(* Visualisation AUTO1
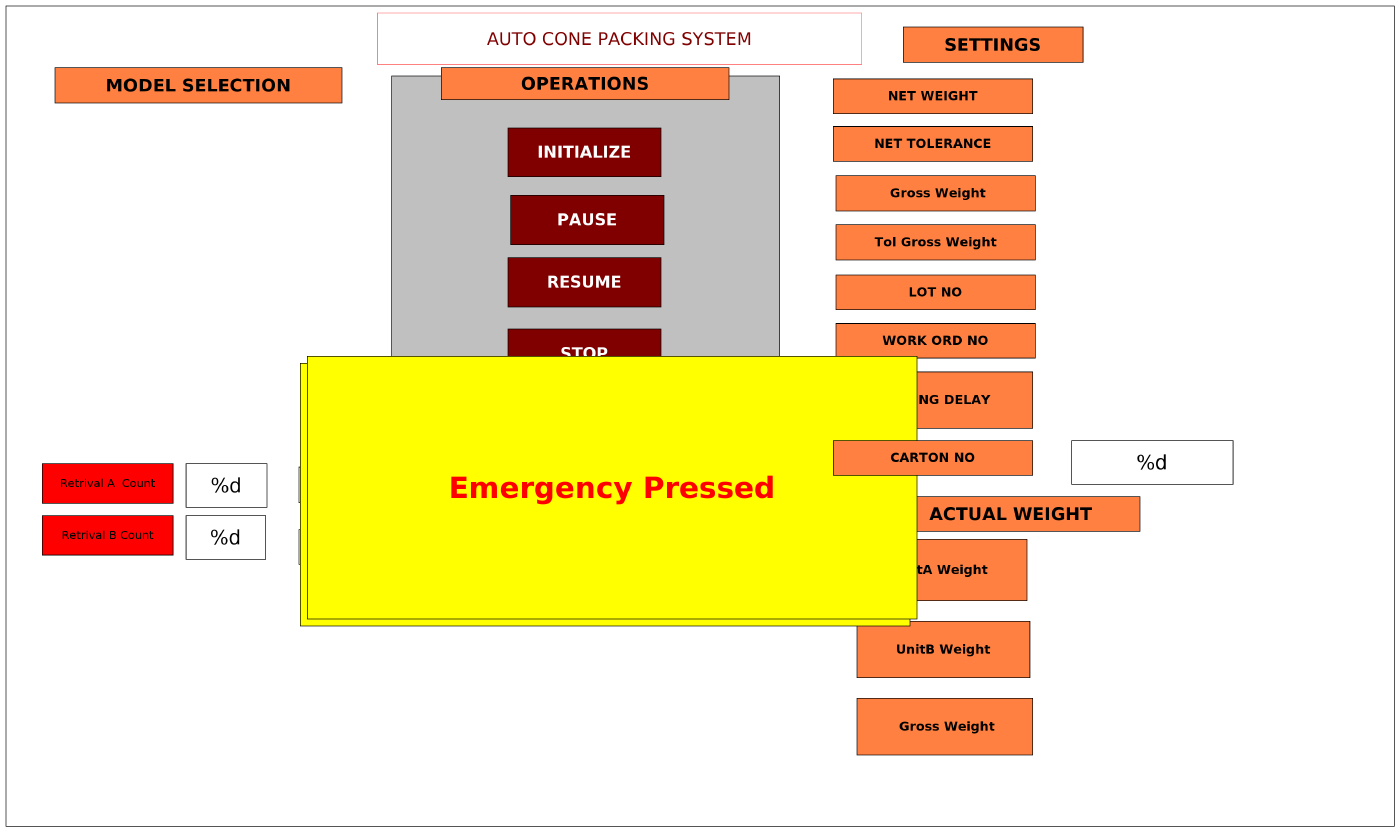
rounded rectangle at (530,10)-(1221,84): text "AUTO CONE PACKING SYSTEM"
rounded rectangle at (418,658)-(674,709): text "Machine Status"
rounded rectangle at (693,648)-(1093,718): text "%s"; shows sAMcModeStatus
rounded rectangle at (418,747)-(674,797): text "Alarm Status"
rounded rectangle at (693,737)-(1093,807): text "%s"; shows sAlarmStatus
rounded rectangle at (70,88)-(480,139): text "MODEL SELECTION"
rounded rectangle at (1210,761)-(1457,849): text "UnitA Weight"
rounded rectangle at (1214,878)-(1461,959): text "UnitB Weight"
rounded rectangle at (1184,522)-(1465,603): text "SEALING DELAY"
rounded rectangle at (1280,30)-(1537,81): text "SETTINGS"
rounded rectangle at (1180,104)-(1465,154): text "NET WEIGHT"
rounded rectangle at (1180,172)-(1465,222): text "NET TOLERANCE"
rounded rectangle at (1249,700)-(1618,750): text "ACTUAL WEIGHT"
rounded rectangle at (257,727)-(371,790): text "%d"; shows UnitBConeCountHMI
rounded rectangle at (257,653)-(373,716): text "%d"; shows UnitAConeCountHMI
rectangle at (52,653)-(239,710): text "Retrival A  Count"
rectangle at (52,727)-(239,784): text "Retrival B Count"
rounded rectangle at (1184,384)-(1469,434): text "LOT NO"
rounded rectangle at (1184,242)-(1469,293): text "Gross Weight"
rounded rectangle at (1214,988)-(1465,1069): text "Gross Weight"
rounded rectangle at (1184,312)-(1469,363): text "Tol Gross Weight"
rounded rectangle at (1184,453)-(1469,503): text "WORK ORD NO"
rounded rectangle at (716,461)-(935,532): text "STOP"; alarm colour if bStopHmi; taps bStopHmi
rounded rectangle at (716,359)-(935,430): text "RESUME"; alarm colour if bAPauseSeq; taps bResumeHmi
rounded rectangle at (720,270)-(939,341): text "PAUSE"; alarm colour if bAPauseSeq; taps bPauseHmi
rounded rectangle at (716,174)-(935,244): text "INITIALIZE"; alarm colour if bAInitializeSeq; taps bInitializeHmi
rounded rectangle at (621,88)-(1032,134): text "OPERATIONS"
rounded rectangle at (420,510)-(1290,885): text "Supply Pressure Low"; invisible if NOT bPrssurePopUp
rounded rectangle at (430,500)-(1300,875): text "Emergency Pressed"; invisible if NOT bEmPopUp
rounded rectangle at (1180,620)-(1465,670): text "CARTON NO"
rounded rectangle at (1520,620)-(1751,683): text "%d"; shows CARTONNO_DIS
2 more shapes without text or variables
20 elements of other kinds (tables, trends, ...) not read
*)

(* Visualisation DIAGNOSTICS
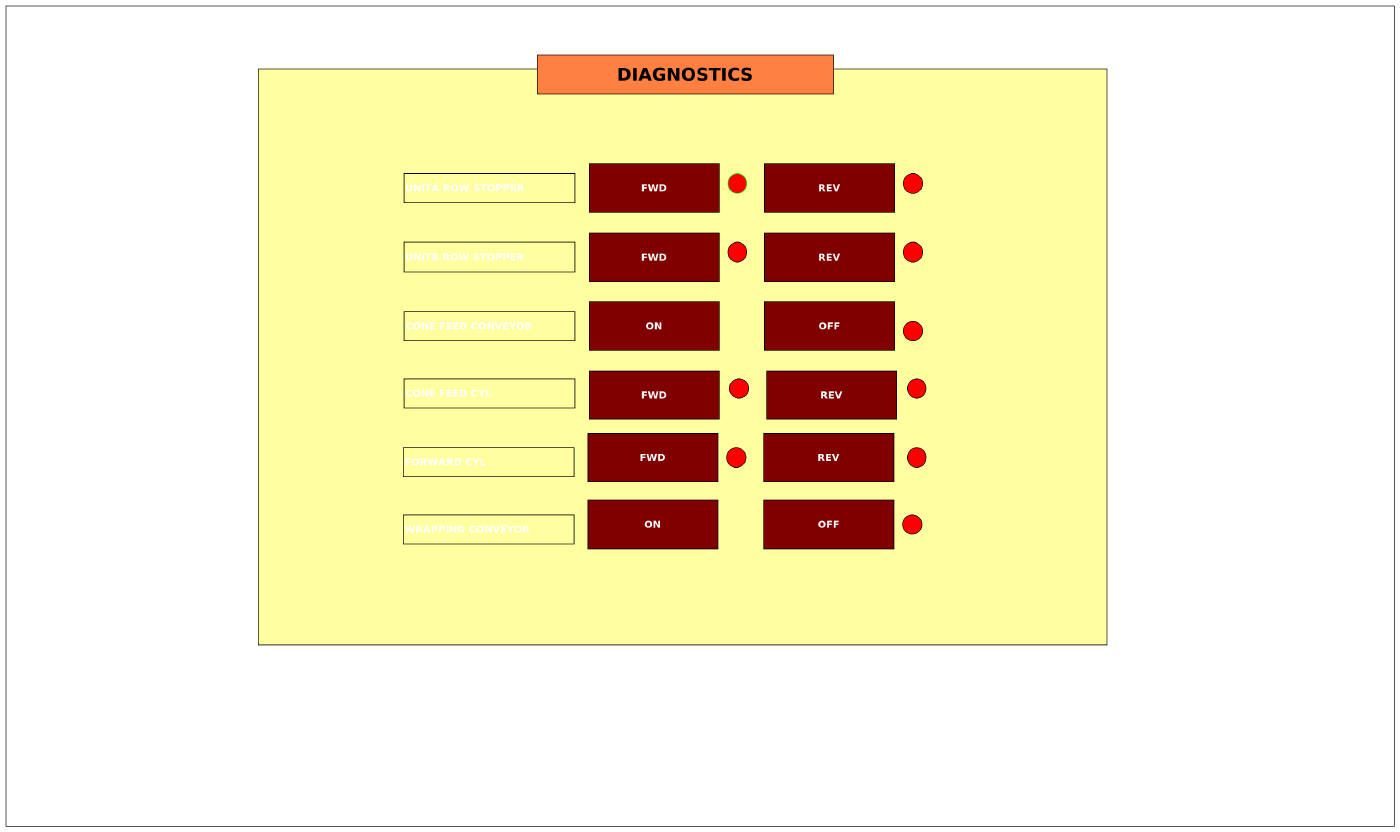
rounded rectangle at (758,70)-(1181,126): text "DIAGNOSTICS"
ellipse at (1030,239)-(1057,268): alarm colour if .bIUnitA_RowStopperEnd
ellipse at (1030,337)-(1057,366): alarm colour if .bIUnitB_RowStopperEnd
ellipse at (1280,239)-(1308,268): alarm colour if .bIUnitA_RowStopperHome
ellipse at (1280,337)-(1308,366): alarm colour if .bIUnitB_RowStopperHome
ellipse at (1280,450)-(1308,478): alarm colour if .bQFeedingConveyorMotor
rounded rectangle at (832,225)-(1018,295): text "FWD"; alarm colour if .bUA_RowStopperMotorFwdOnHmi; taps .bUA_RowStopperMotorFwdOnHmi
rounded rectangle at (1082,225)-(1268,295): text "REV"; alarm colour if .bUA_RowStopperMotorRevOnHmi; taps .bUA_RowStopperMotorRevOnHmi
rounded rectangle at (832,324)-(1018,394): text "FWD"; alarm colour if .bUB_RowStopperMotorFwdOnHmi; taps .bUB_RowStopperMotorFwdOnHmi
rounded rectangle at (832,422)-(1018,492): text "ON"; alarm colour if bFCMotorOnHmi; taps bFCMotorOnHmi
rounded rectangle at (1082,324)-(1268,394): text "REV"; alarm colour if .bUB_RowStopperMotorRevOnHmi; taps .bUB_RowStopperMotorRevOnHmi
rounded rectangle at (1082,422)-(1268,492): text "OFF"; alarm colour if bFCMotorOffHmi; taps bFCMotorOffHmi
rounded rectangle at (568,239)-(812,281): text "UNITA ROW STOPPER"
rounded rectangle at (568,337)-(812,380): text "UNITB ROW STOPPER"
rounded rectangle at (568,436)-(812,478): text "CONE FEED CONVEYOR"
ellipse at (1032,532)-(1060,560): alarm colour if .bIConeFeedingPistonEnd
ellipse at (1286,532)-(1313,560): alarm colour if .bIConeFeedingPistonHome
rounded rectangle at (832,521)-(1018,590): text "FWD"; alarm colour if .bCFPistonOnHmi; taps .bCFPistonOnHmi
rounded rectangle at (1085,521)-(1271,590): text "REV"; alarm colour if .bCFPistonOffHmi; taps .bCFPistonOffHmi
rounded rectangle at (568,532)-(812,574): text "CONE FEED CYL"
ellipse at (1279,726)-(1307,754): alarm colour if .bQMWrappingConveyorMotor
rounded rectangle at (830,705)-(1016,775): text "ON"; alarm colour if .bWCMotorOnHmi; taps .bWCMotorOnHmi
rounded rectangle at (1081,705)-(1267,775): text "OFF"; alarm colour if .bWCMotorOffHmi; taps .bWCMotorOffHmi
rounded rectangle at (567,726)-(811,768): text "WRAPPING CONVEYOR"
rounded rectangle at (567,630)-(811,672): text "FORWARD CYL"
rounded rectangle at (830,610)-(1016,679): text "FWD"; alarm colour if .bFPValveOnHmi; taps .bFPValveOnHmi
rounded rectangle at (1081,610)-(1267,679): text "REV"; alarm colour if .bFPValveOffHmi; taps .bFPValveOffHmi
ellipse at (1028,630)-(1056,659): alarm colour if .bIForwardPistonEnd
ellipse at (1286,630)-(1313,659): alarm colour if .bIForwardPistonHome
2 more shapes without text or variables
2 elements of other kinds (tables, trends, ...) not read
*)

(* Visualisation DIAGNOSTICS_1
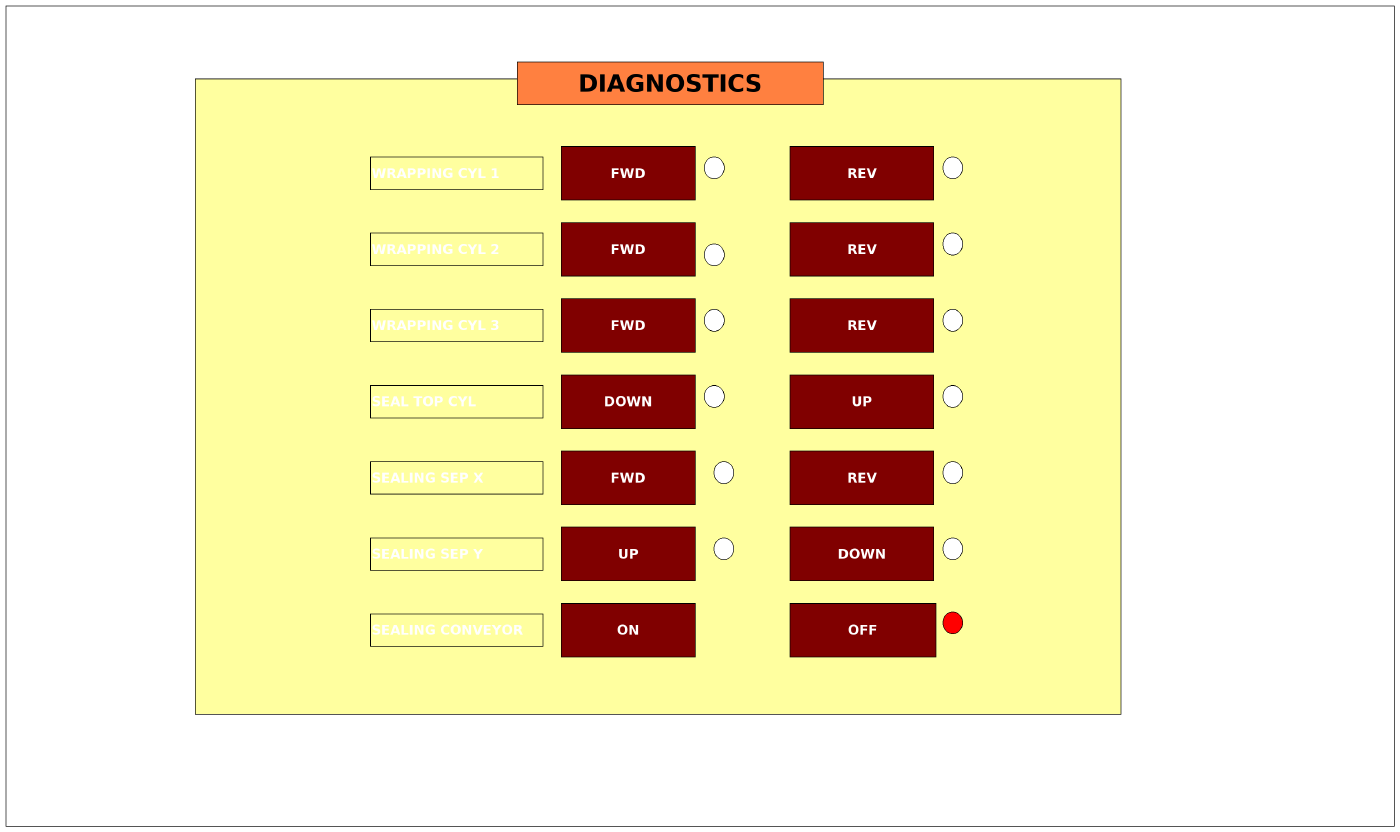
group at (270,80)-(1591,1011)
  rounded rectangle at (338,0)-(659,41): text "DIAGNOSTICS"
  rounded rectangle at (384,80)-(525,131): text "FWD"; alarm colour if .bWrappingCPV1OnHmi; taps .bWrappingCPV1OnHmi
  rounded rectangle at (384,152)-(525,203): text "FWD"; alarm colour if .bWrappingCPV2OnHmi; taps .bWrappingCPV2OnHmi
  rounded rectangle at (624,152)-(775,203): text "REV"; alarm colour if .bWrappingCPV2OffHmi; taps .bWrappingCPV2OffHmi
  rounded rectangle at (384,224)-(525,275): text "FWD"; alarm colour if .bWrappingCPV3OnHmi; taps .bWrappingCPV3OnHmi
  rounded rectangle at (624,224)-(775,275): text "REV"; alarm colour if .bWrappingCPV3OffHmi; taps .bWrappingCPV3OffHmi
  rounded rectangle at (384,296)-(525,347): text "DOWN"; alarm colour if .bSealingTopPVOnHmi; taps .bSealingTopPVOnHmi
  rounded rectangle at (624,296)-(775,347): text "UP"; alarm colour if bSealingTopPVOffHmi; taps bSealingTopPVOffHmi
  rounded rectangle at (384,368)-(525,419): text "FWD"; alarm colour if bSSXAxisPistonValveOnHmi; taps bSSXAxisPistonValveOnHmi
  rounded rectangle at (624,368)-(775,419): text "REV"; alarm colour if bSSXAxisPistonValveOffHmi; taps bSSXAxisPistonValveOffHmi
  rounded rectangle at (184,90)-(365,121): text "WRAPPING CYL 1"
  rounded rectangle at (184,162)-(365,193): text "WRAPPING CYL 2"
  rounded rectangle at (184,234)-(365,265): text "WRAPPING CYL 3"
  rounded rectangle at (184,306)-(365,337): text "SEAL TOP CYL"
  rounded rectangle at (184,378)-(365,409): text "SEALING SEP X"
  rounded rectangle at (624,80)-(775,131): text "REV"; alarm colour if .bWrappingCPV1OffHmi; taps .bWrappingCPV1OffHmi
  ellipse at (784,520)-(805,541): alarm colour if .bQMWrappingConveyorMotor
  rounded rectangle at (384,512)-(525,563): text "ON"; alarm colour if bSCMotorOnHmi; taps bSCMotorOnHmi
  rounded rectangle at (624,512)-(777,563): text "OFF"; alarm colour if bSCMotorOffHmi; taps bSCMotorOffHmi
  rounded rectangle at (184,522)-(365,553): text "SEALING CONVEYOR"
  rounded rectangle at (384,440)-(525,491): text "UP"; alarm colour if bSSYAxisPistonValveOnHmi; taps bSSYAxisPistonValveOnHmi
  rounded rectangle at (624,440)-(775,491): text "DOWN"; alarm colour if bSSYAxisPistonValveOffHmi; taps bSSYAxisPistonValveOffHmi
  rounded rectangle at (184,450)-(365,481): text "SEALING SEP Y"
14 more shapes without text or variables
*)

(* Visualisation OVERVIEW
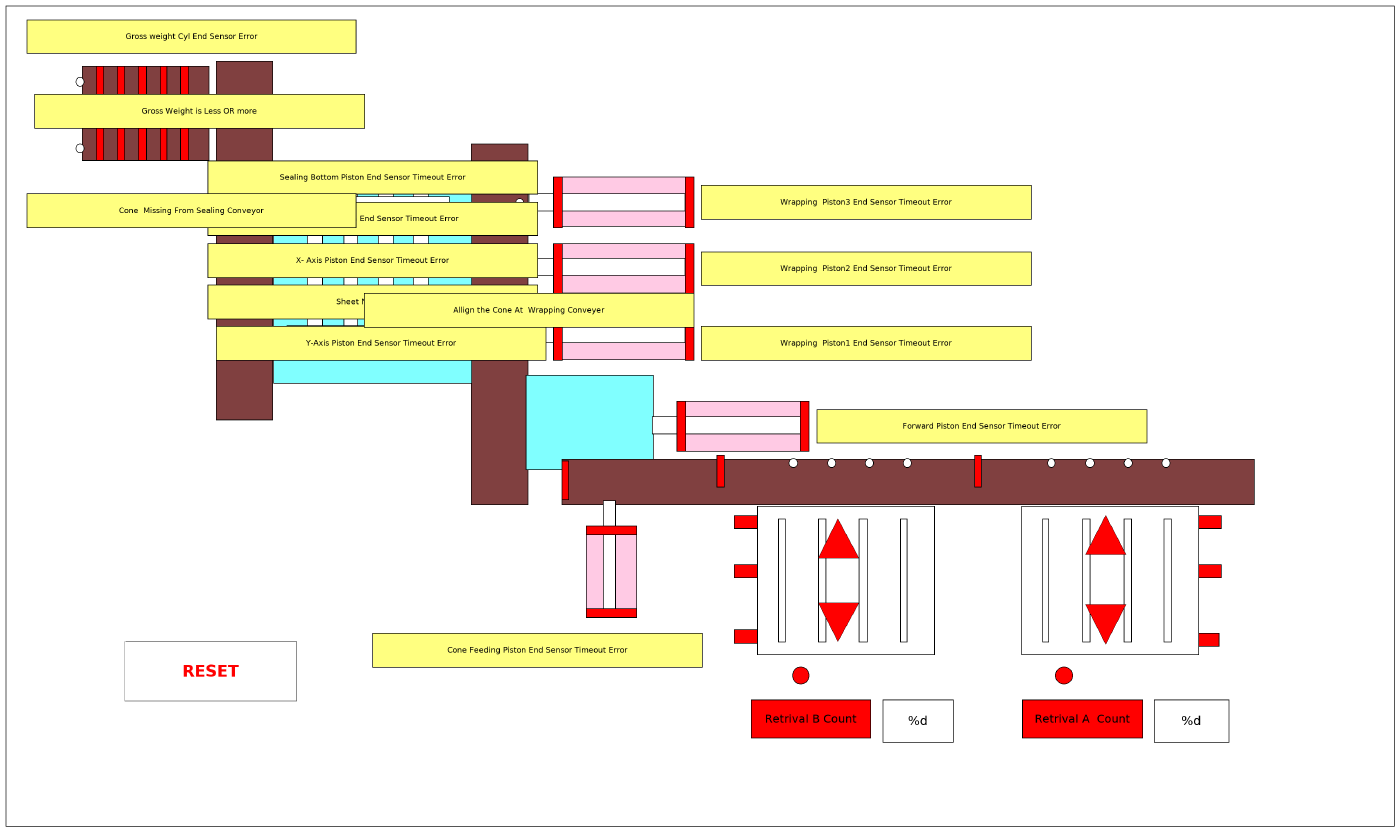
rectangle at (746,360)-(969,385): alarm colour if bQWrappingChannelPistonValve2
rectangle at (781,339)-(794,411): alarm colour if bIWrappingChannelPiston2_End
rectangle at (969,339)-(982,411): alarm colour if bIWrappingChannelPiston2_Home
rectangle at (1685,895)-(1731,914): alarm colour if bIUnitA_RowStopperHome
rectangle at (1692,797)-(1734,816): alarm colour if bIUnitA_RowStopperMiddle
rectangle at (1692,727)-(1734,746): alarm colour if bIUnitA_RowStopperEnd
rectangle at (1039,727)-(1077,746): alarm colour if bIUnitB_RowStopperEnd
rectangle at (1039,890)-(1077,910): alarm colour if bIUnitB_RowStopperHome
rectangle at (1039,797)-(1077,816): alarm colour if bIUnitB_RowStopperMiddle
rounded rectangle at (664,197)-(745,712): alarm colour if bQWrappingConveyorMotor
rectangle at (922,586)-(1144,611): alarm colour if bQForwardPistonValve
rounded rectangle at (793,647)-(1781,712): alarm colour if bQFeedingConveyorMotor
polygon at (1159,852)-(1217,907): alarm colour if bQUnitBRowStopperMotorRev
polygon at (1159,732)-(1217,788): alarm colour if bQUnitBRowStopperMotorFwd
polygon at (1540,854)-(1598,911): alarm colour if bQUnitARowStopperMotorRev
polygon at (1540,727)-(1598,783): alarm colour if bQUnitARowStopperMotorFwd
rectangle at (793,649)-(803,705): alarm colour if bIConeOrientationTop
rectangle at (1014,641)-(1025,687): alarm colour if bIUnitBConeCrossing
rectangle at (1382,641)-(1392,687): alarm colour if bIUnitAConeCrossing
rectangle at (852,706)-(870,872): alarm colour if bQConeFeedingPistonValve
rectangle at (746,457)-(969,481): alarm colour if bQWrappingChannelPistonValve1
rectangle at (746,268)-(969,293): alarm colour if bQWrappingChannelPistonValve3
rectangle at (482,240)-(502,488): alarm colour if bQSealingBottomPistonValve
rectangle at (430,240)-(452,488): alarm colour if bQSealingSeparatorXAxisPistonValve
rectangle at (531,240)-(553,488): alarm colour if bQSealingTopPistonValve
rectangle at (581,244)-(603,494): alarm colour if bQSealingSeparatorYAxisPistonValve
rounded rectangle at (300,79)-(381,591): alarm colour if bQSealingConveyorMotorFWD
rectangle at (109,86)-(290,221): alarm colour if bQGross_Cylinder_On
rectangle at (220,86)-(230,221): alarm colour if bQGross_Roller_On
rectangle at (249,86)-(261,221): alarm colour if bQGross_Roller_On
rectangle at (189,86)-(201,221): alarm colour if bQGross_Roller_On
rectangle at (159,86)-(170,221): alarm colour if bQGross_Roller_On
rectangle at (129,86)-(140,221): alarm colour if bQGross_Roller_On
rectangle at (401,456)-(633,478): alarm colour if bQFilmRollerMotor1
rectangle at (401,272)-(633,292): alarm colour if bQFilmRollerMotor3
rectangle at (401,363)-(633,385): alarm colour if bQFilmRollerMotor2
ellipse at (1540,646)-(1553,659): alarm colour if bIUnitAConeDetection3
ellipse at (1595,646)-(1607,659): alarm colour if bIUnitAConeDetection2
ellipse at (1649,646)-(1661,659): alarm colour if bIUnitAConeDetection1
ellipse at (1486,646)-(1497,659): alarm colour if bIUnitAConeDetection4
ellipse at (1172,646)-(1184,659): alarm colour if bIUnitBConeDetection3
ellipse at (1226,646)-(1238,659): alarm colour if bIUnitBConeDetection2
ellipse at (1280,646)-(1292,659): alarm colour if bIUnitBConeDetection1
ellipse at (1117,646)-(1130,659): alarm colour if bIUnitBConeDetection4
ellipse at (727,275)-(739,288): alarm colour if bIWrappingCone3
ellipse at (727,368)-(739,381): alarm colour if bIWrappingCone2
ellipse at (722,457)-(734,470): alarm colour if bIWrappingCone1
ellipse at (327,229)-(338,241): alarm colour if bIConeCountSensor
ellipse at (597,221)-(608,233): alarm colour if bISealingSeparatorYAxisEnd
ellipse at (441,221)-(453,233): alarm colour if bISealingSeparatorXAxisEnd
ellipse at (553,221)-(565,233): alarm colour if bISealingTopPistonEnd
ellipse at (499,221)-(511,233): alarm colour if bISealingBottomPistonEnd
ellipse at (100,102)-(112,115): alarm colour if bIGross_Cyl_Home
ellipse at (100,197)-(112,210): alarm colour if bIGross_Cyl_End
ellipse at (1122,943)-(1146,968): alarm colour if bQUnitBWeightOkLamp
ellipse at (1497,943)-(1522,968): alarm colour if bQUnitAWeightOkLamp
rectangle at (781,244)-(794,317): alarm colour if bIWrappingChannelPiston3_End
rectangle at (969,244)-(982,317): alarm colour if bIWrappingChannelPiston3_Home
rectangle at (781,434)-(794,506): alarm colour if bIWrappingChannelPiston1_End
rectangle at (969,434)-(982,506): alarm colour if bIWrappingChannelPiston1_Home
rectangle at (828,742)-(900,755): alarm colour if bIConeFeedingPistonEnd
rectangle at (828,860)-(900,873): alarm colour if bIConeFeedingPistonHome
rectangle at (1133,564)-(1146,636): alarm colour if bIForwardPistonHome
ellipse at (592,493)-(605,506): alarm colour if bISealingSeparatorYAxisHome
ellipse at (441,493)-(452,506): alarm colour if bISealingSeparatorXAxisHome
ellipse at (549,493)-(561,506): alarm colour if bISealingTopPistonHome
ellipse at (495,493)-(506,506): alarm colour if bISealingBottomPistonHome
rectangle at (523,895)-(994,944): text "Cone Feeding Piston End Sensor Timeout Error"; invisible if NOT bAConeFeedCylRsError
rectangle at (992,457)-(1463,506): text "Wrapping  Piston1 End Sensor Timeout Error"; invisible if NOT bAWrappingCylRs1Error
rectangle at (992,256)-(1463,305): text "Wrapping  Piston3 End Sensor Timeout Error"; invisible if NOT bAWrappingCylRs3Error
rectangle at (992,351)-(1463,399): text "Wrapping  Piston2 End Sensor Timeout Error"; invisible if NOT bAWrappingCylRs2Error
rectangle at (288,221)-(759,269): text "Sealing Bottom Piston End Sensor Timeout Error"; invisible if NOT bASealBotCylRsError
rectangle at (288,280)-(759,328): text "Sealing Top Piston End Sensor Timeout Error"; invisible if NOT bASealTopCylRsError
rectangle at (288,339)-(759,388): text "X- Axis Piston End Sensor Timeout Error"; invisible if NOT bASealSepXCylRsError
rectangle at (300,457)-(771,506): text "Y-Axis Piston End Sensor Timeout Error"; invisible if NOT bASealSepYCylRsError
rectangle at (288,398)-(759,447): text "Sheet NOT Feeded"; invisible if NOT bAPolythinSheetError
rectangle at (30,268)-(500,317): text "Cone  Missing From Sealing Conveyor"; invisible if NOT bAConeMissAtSealConv
rectangle at (511,410)-(982,459): text "Allign the Cone At  Wrapping Conveyer"; invisible if NOT bAConeMissErrorAtWrpConv
rectangle at (41,126)-(512,175): text "Gross Weight is Less OR more"; invisible if NOT bGrossWieghtNOk
rectangle at (1157,576)-(1628,624): text "Forward Piston End Sensor Timeout Error"; invisible if NOT bAFwdCylRsError
rectangle at (30,20)-(500,68): text "Gross weight Cyl End Sensor Error"; invisible if NOT bGrossWtCylEndSenError
button at (170,907)-(415,992): text "RESET"; shows .bErrorReset; taps .bErrorResethmi
rounded rectangle at (1251,990)-(1352,1051): text "%d"; shows UnitBConeCountHMI
rounded rectangle at (1638,990)-(1745,1051): text "%d"; shows UnitAConeCountHMI_1
rectangle at (1450,990)-(1622,1045): text "Retrival A  Count"
rectangle at (1063,990)-(1234,1045): text "Retrival B Count"
19 more shapes without text or variables
6 elements of other kinds (tables, trends, ...) not read
*)

(* Visualisation PARAMETERS
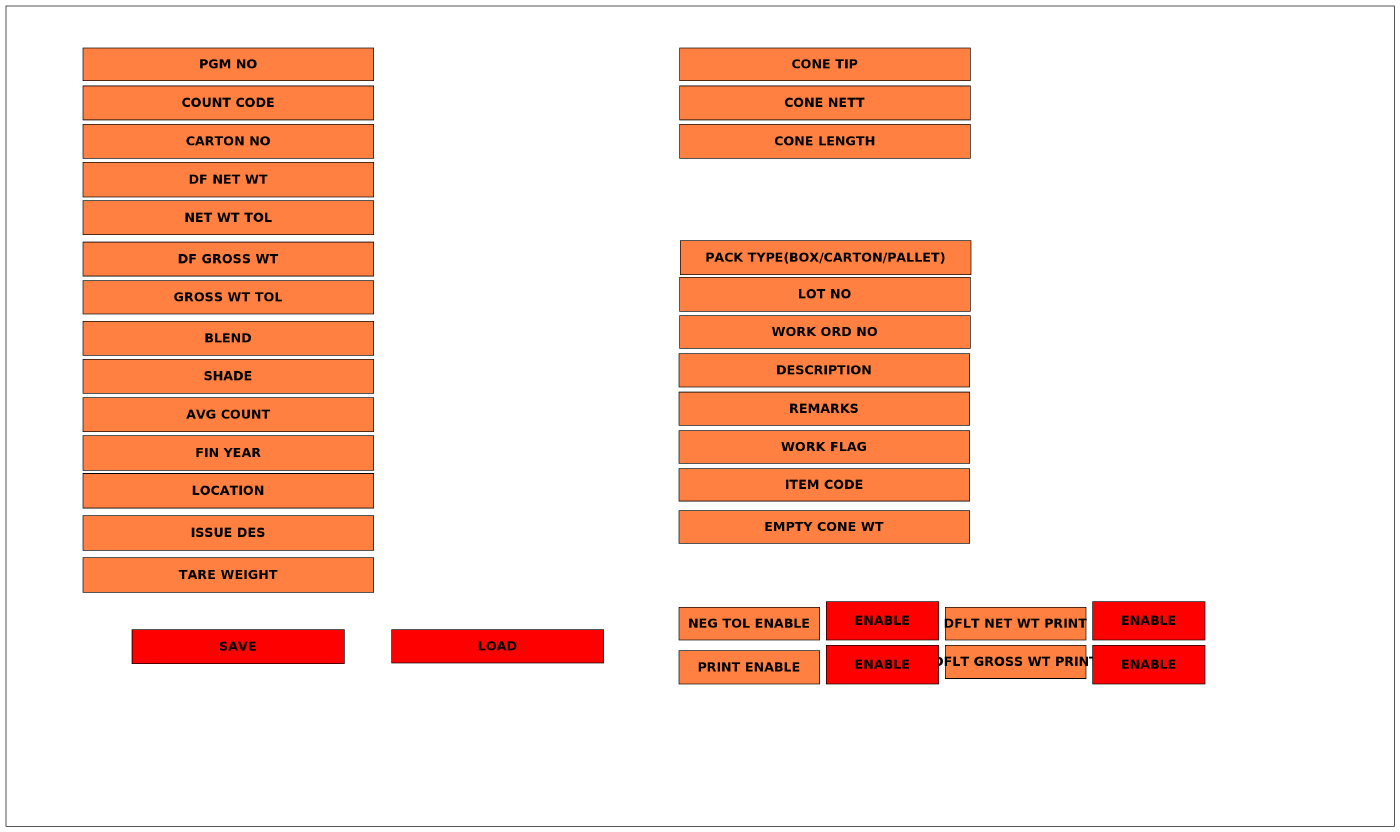
rounded rectangle at (110,60)-(525,107): text "PGM NO"
rounded rectangle at (110,114)-(525,163): text "COUNT CODE"
rounded rectangle at (110,223)-(525,273): text "DF NET WT"
rounded rectangle at (110,169)-(525,218): text "CARTON NO"
rounded rectangle at (110,337)-(525,386): text "DF GROSS WT"
rounded rectangle at (110,450)-(525,499): text "BLEND"
rounded rectangle at (110,504)-(525,553): text "SHADE"
rounded rectangle at (961,60)-(1376,107): text "CONE TIP"
rounded rectangle at (961,114)-(1376,163): text "CONE NETT"
rounded rectangle at (961,169)-(1376,218): text "CONE LENGTH"
rounded rectangle at (962,335)-(1377,384): text "PACK TYPE(BOX/CARTON/PALLET)"
rounded rectangle at (961,387)-(1376,436): text "LOT NO"
rounded rectangle at (961,442)-(1376,489): text "WORK ORD NO"
rounded rectangle at (180,890)-(483,939): text "SAVE"; alarm colour if SAVE; taps SAVE
rounded rectangle at (550,890)-(853,938): text "LOAD"; opens PARAMETERS_LOAD
rounded rectangle at (110,278)-(525,327): text "NET WT TOL"
rounded rectangle at (110,392)-(525,440): text "GROSS WT TOL"
rounded rectangle at (960,858)-(1161,905): text "NEG TOL ENABLE"
rounded rectangle at (1170,850)-(1331,905): text "ENABLE"; alarm colour if NegTolEnableHmi; toggles NegTolEnableHmi
rounded rectangle at (1340,858)-(1541,905): text "DFLT NET WT PRINT"
rounded rectangle at (1340,912)-(1541,960): text "DFLT GROSS WT PRINT"
rounded rectangle at (1550,850)-(1711,905): text "ENABLE"; alarm colour if DfltWtPrint; toggles DfltWtPrint
rounded rectangle at (1550,912)-(1711,968): text "ENABLE"; alarm colour if GrossWtPrintDflt; toggles GrossWtPrintDflt
rounded rectangle at (960,920)-(1161,968): text "PRINT ENABLE"
rounded rectangle at (1170,912)-(1331,968): text "ENABLE"; alarm colour if PrintEnableHmi; toggles PrintEnableHmi
rounded rectangle at (110,559)-(525,608): text "AVG COUNT"
rounded rectangle at (110,613)-(525,663): text "FIN YEAR"
rounded rectangle at (960,496)-(1375,544): text "DESCRIPTION"
rounded rectangle at (960,551)-(1375,599): text "REMARKS"
rounded rectangle at (960,606)-(1375,653): text "WORK FLAG"
rounded rectangle at (110,667)-(525,717): text "LOCATION"
rounded rectangle at (960,660)-(1375,707): text "ITEM CODE"
rounded rectangle at (110,727)-(525,777): text "ISSUE DES"
rounded rectangle at (960,720)-(1375,767): text "EMPTY CONE WT"
rounded rectangle at (110,787)-(525,837): text "TARE WEIGHT"
1 more shapes without text or variables
32 elements of other kinds (tables, trends, ...) not read
*)

(* Visualisation PARAMETERS_LOAD
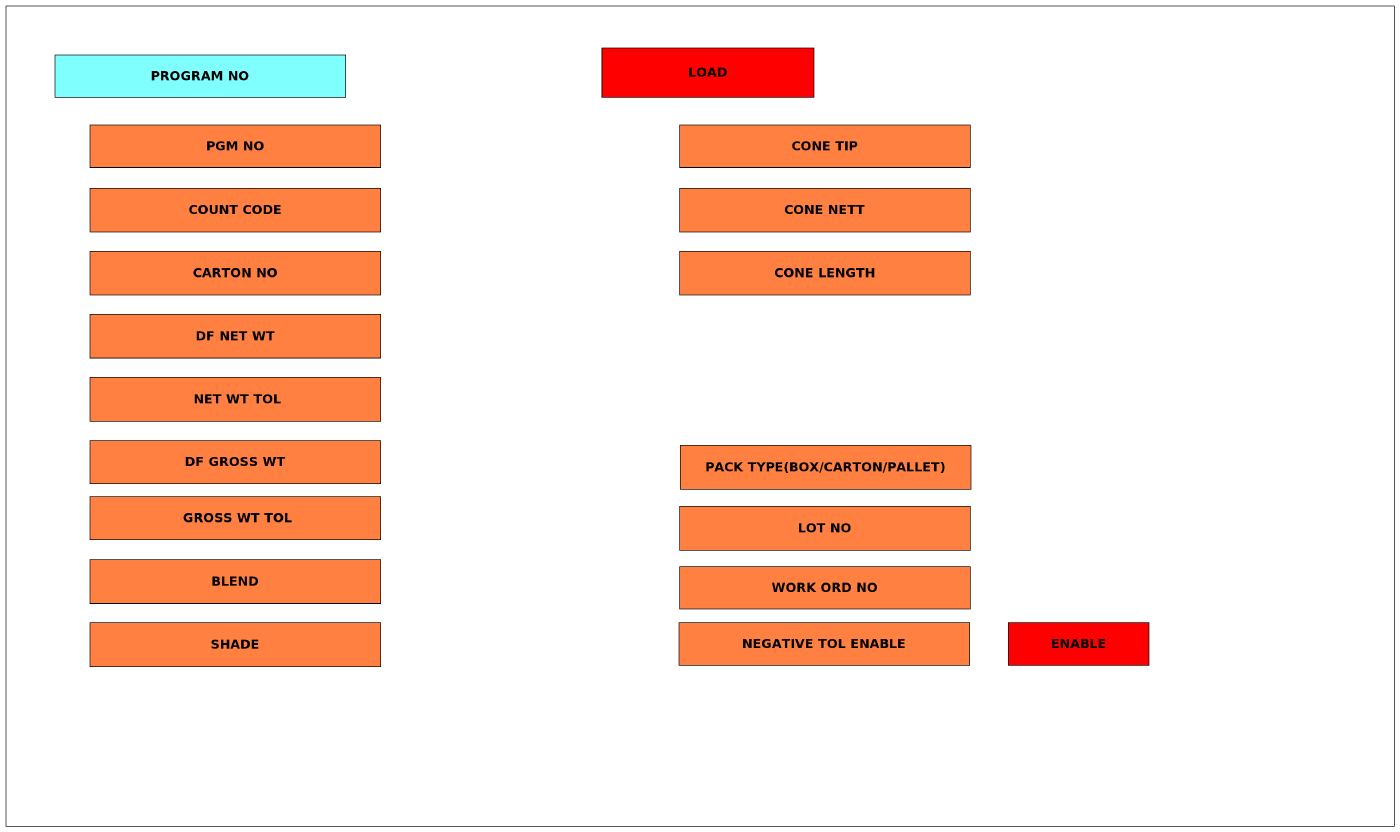
rounded rectangle at (120,170)-(535,231): text "PGM NO"
rounded rectangle at (120,260)-(535,323): text "COUNT CODE"
rounded rectangle at (120,440)-(535,503): text "DF NET WT"
rounded rectangle at (120,350)-(535,413): text "CARTON NO"
rounded rectangle at (120,620)-(535,682): text "DF GROSS WT"
rounded rectangle at (120,790)-(535,853): text "BLEND"
rounded rectangle at (120,880)-(535,943): text "SHADE"
rounded rectangle at (961,170)-(1376,231): text "CONE TIP"
rounded rectangle at (961,260)-(1376,323): text "CONE NETT"
rounded rectangle at (961,350)-(1376,413): text "CONE LENGTH"
rounded rectangle at (962,627)-(1377,690): text "PACK TYPE(BOX/CARTON/PALLET)"
rounded rectangle at (961,714)-(1376,777): text "LOT NO"
rounded rectangle at (961,800)-(1376,861): text "WORK ORD NO"
rounded rectangle at (70,70)-(485,131): text "PROGRAM NO"
rounded rectangle at (850,60)-(1153,131): text "LOAD"; alarm colour if LOAD; taps LOAD
rounded rectangle at (120,530)-(535,593): text "NET WT TOL"
rounded rectangle at (120,700)-(535,762): text "GROSS WT TOL"
rounded rectangle at (960,880)-(1375,941): text "NEGATIVE TOL ENABLE"
rounded rectangle at (1430,880)-(1631,941): text "ENABLE"; alarm colour if negativetolerance; taps NegTolEnableHmi
1 more shapes without text or variables
23 elements of other kinds (tables, trends, ...) not read
*)

(* Visualisation PARAMETERS_OVERVIEW
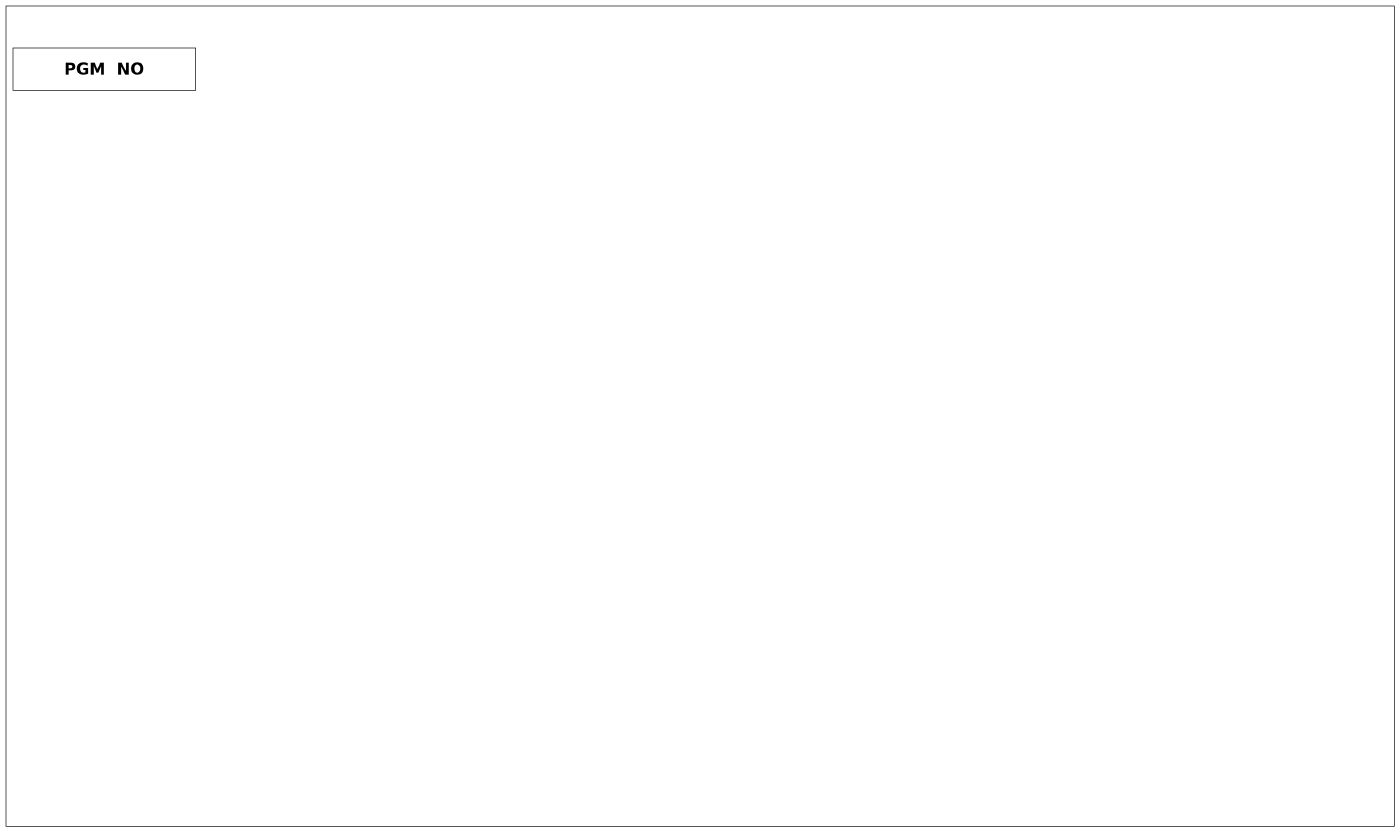
rectangle at (10,60)-(271,121): text "PGM  NO"
1 more shapes without text or variables
*)
